# EPICS substitutions: ecmcApp/Db/SolAxis-extra.substitutions
file "ecmc-extra.template"
{
pattern
{P,      M,    R,   PORT, ADDR, PREC, HOMEPROC}
{IOC2:,  m1, m1-,   MCU1,    1, 3,    3}
}
